{attribute 'linkalways'} 
{attribute 'no_explicit_call' := 'This FB is a CLASS and must be accessed using methods or properties'}
{attribute 'enable_dynamic_creation'}
FUNCTION_BLOCK FINAL LT_ULINT EXTENDS Node
VAR
	in1 : _ULINT(0);
	in2 : _ULINT(0);
	out : _BOOL(FALSE);
END_VAR

METHOD PUBLIC Clone : I_Node
VAR
	pNode : POINTER TO LT_ULINT;
END_VAR
pNode := __NEW(LT_ULINT);
Clone := pNode^;
END_METHOD

METHOD FB_init : BOOL
VAR_INPUT
	bInitRetains : BOOL; // if TRUE, the retain variables are initialized (warm start / cold start)
	bInCopyCode : BOOL;  // if TRUE, the instance afterwards gets moved into the copy code (online change)
END_VAR
AddInput('in1',THIS^.in1);
AddInput('in2',THIS^.in2);
AddOutput('out', THIS^.out);
END_METHOD

METHOD PROTECTED OnExecute
VAR
END_VAR
out.Value := in1.Value < in2.Value;
END_METHOD

END_FUNCTION_BLOCK

(* stored: Version 1.1.0.1, ProductVersion 3.1.4024.15
   POU LT_ULINT: Id {60cb526b-31b9-45e8-9325-0b24f9cb39ff}, SpecialFunc None
   Folder Constructor: Id {a7b8018e-9d42-4e75-a87a-b3eeb23c2e3c}
   Method Clone: Id {4835c9d3-55f2-43ec-bc09-630823d6f26b}
   Method FB_init: Id {b47d2069-58cf-4e41-9385-633fa2f38514}
   Method OnExecute: Id {ba7b99df-33d0-4825-bd07-56ba1039a6f3} *)
